// TIA Portal project "m1-5s-2s-0c-1t" (V16)

(* hardware
DEVICE "S7-1200 station_1"  S7-1200 Station
   slot 0: "Rack_0"  S7-1200 Rack  Rack  V1.0
   slot 1: "PLC_1"  CPU 1212C AC/DC/Rly  6ES7 212-1BE40-0XB0  V4.0
*)

// ===== PLC "PLC_1"  CPU 1212C AC/DC/Rly =====

VAR_GLOBAL   // PLC tag table "Default tag table"
   "start" AT %I0.0 : Bool;
   "m1" AT %Q0.0 : Bool;
   "timer loop" AT %M0.0 : Bool;
   "timer loop 2" AT %M0.1 : Bool;
   "Tag_1" AT %M0.5 : Bool;
   "stop" AT %I0.1 : Bool;
   "Tag_3" AT %M0.3 : Bool;
   "Tag_2" AT %M0.6 : Bool;
   "Tag_4" AT %M0.4 : Bool;
   "Tag_5" AT %M0.7 : Bool;
   "Tag_6" AT %M1.0 : Bool;
   "Tag_7" AT %M1.1 : Bool;
   "Tag_8" AT %M0.2 : Bool;
   "Tag_9" AT %M1.2 : Bool;
END_VAR

// folder: System blocks/Program resources

DATA_BLOCK "T1"   // DB1
{ S7_Optimized_Access := 'TRUE' }
AUTHOR : Simatic
FAMILY : IEC
NAME : IEC_TMR
VERSION : 1.0
// stored: InstanceOfName IEC_TIMER
"IEC_TIMER"
BEGIN
END_DATA_BLOCK

DATA_BLOCK "C1"   // DB2
{ S7_Optimized_Access := 'TRUE' }
AUTHOR : Simatic
FAMILY : IEC
NAME : CNTR
VERSION : 1.0
// stored: InstanceOfName IEC_COUNTER
"IEC_COUNTER"
BEGIN
END_DATA_BLOCK

DATA_BLOCK "C2"   // DB4
{ S7_Optimized_Access := 'TRUE' }
AUTHOR : Simatic
FAMILY : IEC
NAME : CNTR
VERSION : 1.0
// stored: InstanceOfName IEC_COUNTER
"IEC_COUNTER"
BEGIN
END_DATA_BLOCK

// folder: (top level)

ORGANIZATION_BLOCK "Main"   // OB1, LAD, ProgramCycle
TITLE = "Main Program Sweep (Cycle)"
{ S7_Optimized_Access := 'TRUE' }
VERSION : 0.1
   VAR_INPUT
      Initial_Call : Bool;   // Initial call of this OB
      Remanence : Bool;   // =True, if remanent data are available
   END_VAR
   VAR_TEMP   // added for the SCL form of the ladder/FBD networks
      _w1 : Bool;
      _w2 : Bool;
   END_VAR
BEGIN

REGION Network 1
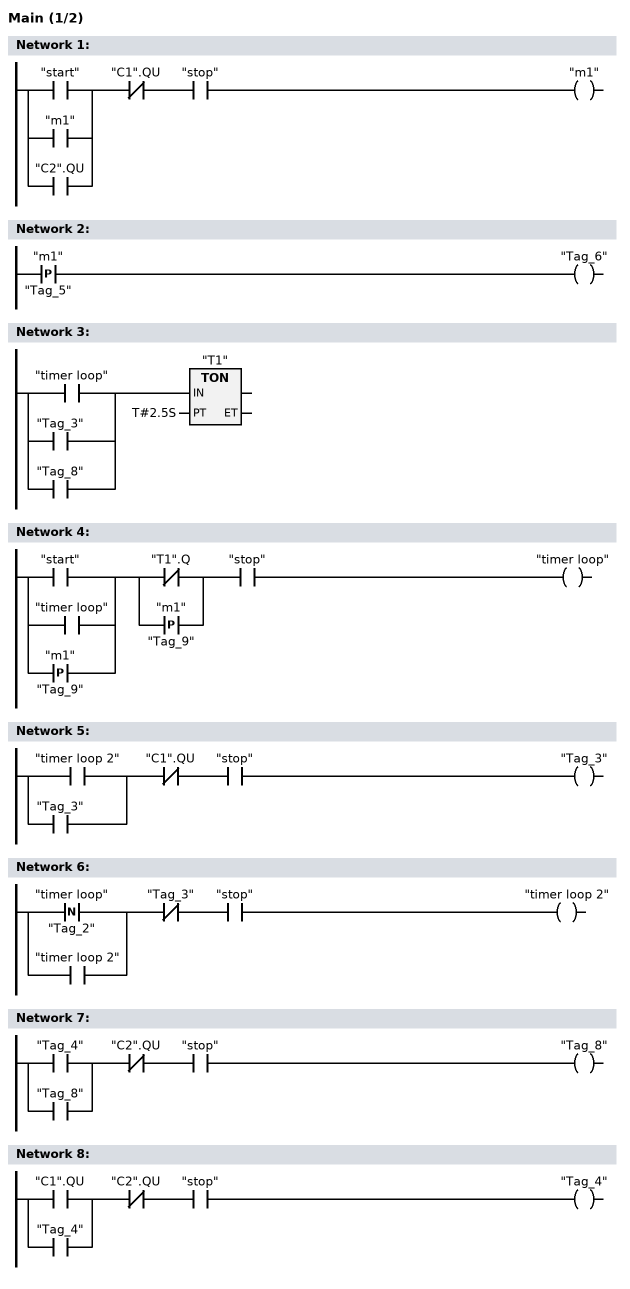
   RUNG wire#powerrail
      Contact( "start" )
      wire#w1
      I_Contact( "C1".QU )
      Contact( "stop" )
      Coil( "m1" )
   END_RUNG
   RUNG wire#powerrail
      Contact( "m1" )
   END_RUNG wire#w1
   RUNG wire#powerrail
      Contact( "C2".QU )
   END_RUNG wire#w1
   // the same network as SCL:
   "m1" := ("start" OR "m1" OR "C2".QU) AND NOT "C1".QU AND "stop";
END_REGION

REGION Network 2
   RUNG wire#powerrail
      P_Contact(operand := "m1", bit := "Tag_5")
      Coil( "Tag_6" )
   END_RUNG
   // the same network as SCL:
   #_w1 := "m1" AND NOT "Tag_5";   // rising edge of "m1"
   "Tag_5" := "m1";
   "Tag_6" := #_w1;
END_REGION

REGION Network 3
   "T1".TON(IN := "timer loop" OR "Tag_3" OR "Tag_8", PT := T#2.5S);
END_REGION

REGION Network 4
   RUNG wire#powerrail
      Contact( "start" )
      wire#w1
      I_Contact( "T1".Q )
      wire#w2
      Contact( "stop" )
      Coil( "timer loop" )
   END_RUNG
   RUNG wire#powerrail
      Contact( "timer loop" )
   END_RUNG wire#w1
   RUNG wire#powerrail
      P_Contact(operand := "m1", bit := "Tag_9")
   END_RUNG wire#w1
   RUNG wire#w1
      P_Contact(operand := "m1", bit := "Tag_9")
   END_RUNG wire#w2
   // the same network as SCL:
   #_w1 := "m1" AND NOT "Tag_9";   // rising edge of "m1"
   "Tag_9" := "m1";
   #_w2 := ("start" OR "timer loop" OR #_w1) AND "m1" AND NOT "Tag_9";   // rising edge of "m1"
   "Tag_9" := "m1";
   "timer loop" := ((("start" OR "timer loop" OR #_w1) AND NOT "T1".Q) OR #_w2) AND "stop";
END_REGION

REGION Network 5
   RUNG wire#powerrail
      Contact( "timer loop 2" )
      wire#w1
      I_Contact( "C1".QU )
      Contact( "stop" )
      Coil( "Tag_3" )
   END_RUNG
   RUNG wire#powerrail
      Contact( "Tag_3" )
   END_RUNG wire#w1
   // the same network as SCL:
   "Tag_3" := ("timer loop 2" OR "Tag_3") AND NOT "C1".QU AND "stop";
END_REGION

REGION Network 6
   RUNG wire#powerrail
      N_Contact(operand := "timer loop", bit := "Tag_2")
      wire#w1
      I_Contact( "Tag_3" )
      Contact( "stop" )
      Coil( "timer loop 2" )
   END_RUNG
   RUNG wire#powerrail
      Contact( "timer loop 2" )
   END_RUNG wire#w1
   // the same network as SCL:
   #_w1 := NOT "timer loop" AND "Tag_2";   // falling edge of "timer loop"
   "Tag_2" := "timer loop";
   "timer loop 2" := (#_w1 OR "timer loop 2") AND NOT "Tag_3" AND "stop";
END_REGION

REGION Network 7
   RUNG wire#powerrail
      Contact( "Tag_4" )
      wire#w1
      I_Contact( "C2".QU )
      Contact( "stop" )
      Coil( "Tag_8" )
   END_RUNG
   RUNG wire#powerrail
      Contact( "Tag_8" )
   END_RUNG wire#w1
   // the same network as SCL:
   "Tag_8" := ("Tag_4" OR "Tag_8") AND NOT "C2".QU AND "stop";
END_REGION

REGION Network 8
   RUNG wire#powerrail
      Contact( "C1".QU )
      wire#w1
      I_Contact( "C2".QU )
      Contact( "stop" )
      Coil( "Tag_4" )
   END_RUNG
   RUNG wire#powerrail
      Contact( "Tag_4" )
   END_RUNG wire#w1
   // the same network as SCL:
   "Tag_4" := ("C1".QU OR "Tag_4") AND NOT "C2".QU AND "stop";
END_REGION

REGION Network 9
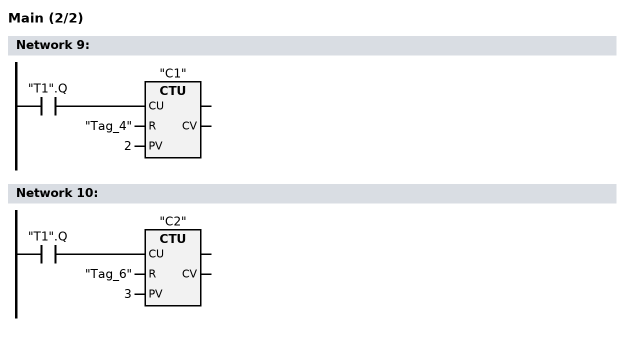
   "C1".CTU(CU := "T1".Q, R := "Tag_4", PV := 2);
END_REGION

REGION Network 10
   "C2".CTU(CU := "T1".Q, R := "Tag_6", PV := 3);
END_REGION
END_ORGANIZATION_BLOCK